// TIA Portal V17 export
// export: Created 2022-02-03T14:45:11.9025904Z, ExportSetting WithDefaults, DisplayName Totally Integrated Automation Portal, DisplayVersion V17, DisplayName TIA Portal Openness, DisplayVersion V17, DisplayName TIA Portal Version Control Interface, DisplayVersion V17, DisplayName SINAMICS Startdrive Advanced, DisplayVersion V17, DisplayName SINAMICS Startdrive G130, G150, S120, S150, SINAMICS MV, S210, DisplayVersion V17, DisplayName SINAMICS Startdrive G110M, G120, G120C, G120D, G120P, G115D, DisplayVersion V17, DisplayName STEP 7 Professional, DisplayVersion V17, DisplayName STEP 7 Safety, DisplayVersion V17, DisplayName WinCC Advanced, DisplayVersion V17
DATA_BLOCK "InstLGF_Frequency"   // DB5
AUTHOR : Siemens_Industry_Support
FAMILY : LGF
NAME : LGF_Frequency
VERSION : 0.1
// stored: Access Unpublished, AutoNumber true, DBAccessibleFromOPCUA true, DBAccessibleFromWebserver true, InstanceOfName LGF_Frequency, InstanceOfType FB
"LGF_Frequency"
   // VAR_INPUT
   //    frequency : Real;
   //    pulsePauseRatio : Real;
   // END_VAR
   // VAR_OUTPUT
   //    clock { ExternalWritable := 'False'} : Bool;
   //    countdown { ExternalWritable := 'False'} : Time;
   // END_VAR
   // VAR
   //    instTofTimePulse { ExternalAccessible := 'False'; ExternalVisible := 'False'; ExternalWritable := 'False'} : TOF_TIME;
   //    instTofTimePause { ExternalAccessible := 'False'; ExternalVisible := 'False'; ExternalWritable := 'False'} : TOF_TIME;
   //    statFrequencyOld { ExternalAccessible := 'False'; ExternalVisible := 'False'; ExternalWritable := 'False'} : Real;
   //    statPulsePauseRatioOld { ExternalAccessible := 'False'; ExternalVisible := 'False'; ExternalWritable := 'False'} : Real;
   //    statTimePulse { ExternalAccessible := 'False'; ExternalVisible := 'False'; ExternalWritable := 'False'} : Time;
   //    statTimePause { ExternalAccessible := 'False'; ExternalVisible := 'False'; ExternalWritable := 'False'} : Time;
   // END_VAR
BEGIN
END_DATA_BLOCK
